PROGRAM SP3_1_Y130
VAR
	CompareOutput130_00: CMP_OC_DW;
	CompareOutput130_01: CMP_OC_DW;
	CompareOutput130_02: CMP_OC_DW;
	CompareOutput130_03: CMP_OC_DW;
	CompareOutput130_04: CMP_OC_DW;
	CompareOutput130_05: CMP_OC_DW;
	CompareOutput130_06: CMP_OC_DW;
	CompareOutput130_07: CMP_OC_DW;
	CompareOutput130_08: CMP_OC_DW;
	CompareOutput130_09: CMP_OC_DW;
	CompareOutput130_10: CMP_OC_DW;
	CompareOutput130_11: CMP_OC_DW;
	CompareOutput130_12: CMP_OC_DW;
	CompareOutput130_13: CMP_OC_DW;
	CompareOutput130_14: CMP_OC_DW;
	CompareOutput130_15: CMP_OC_DW;

END_VAR

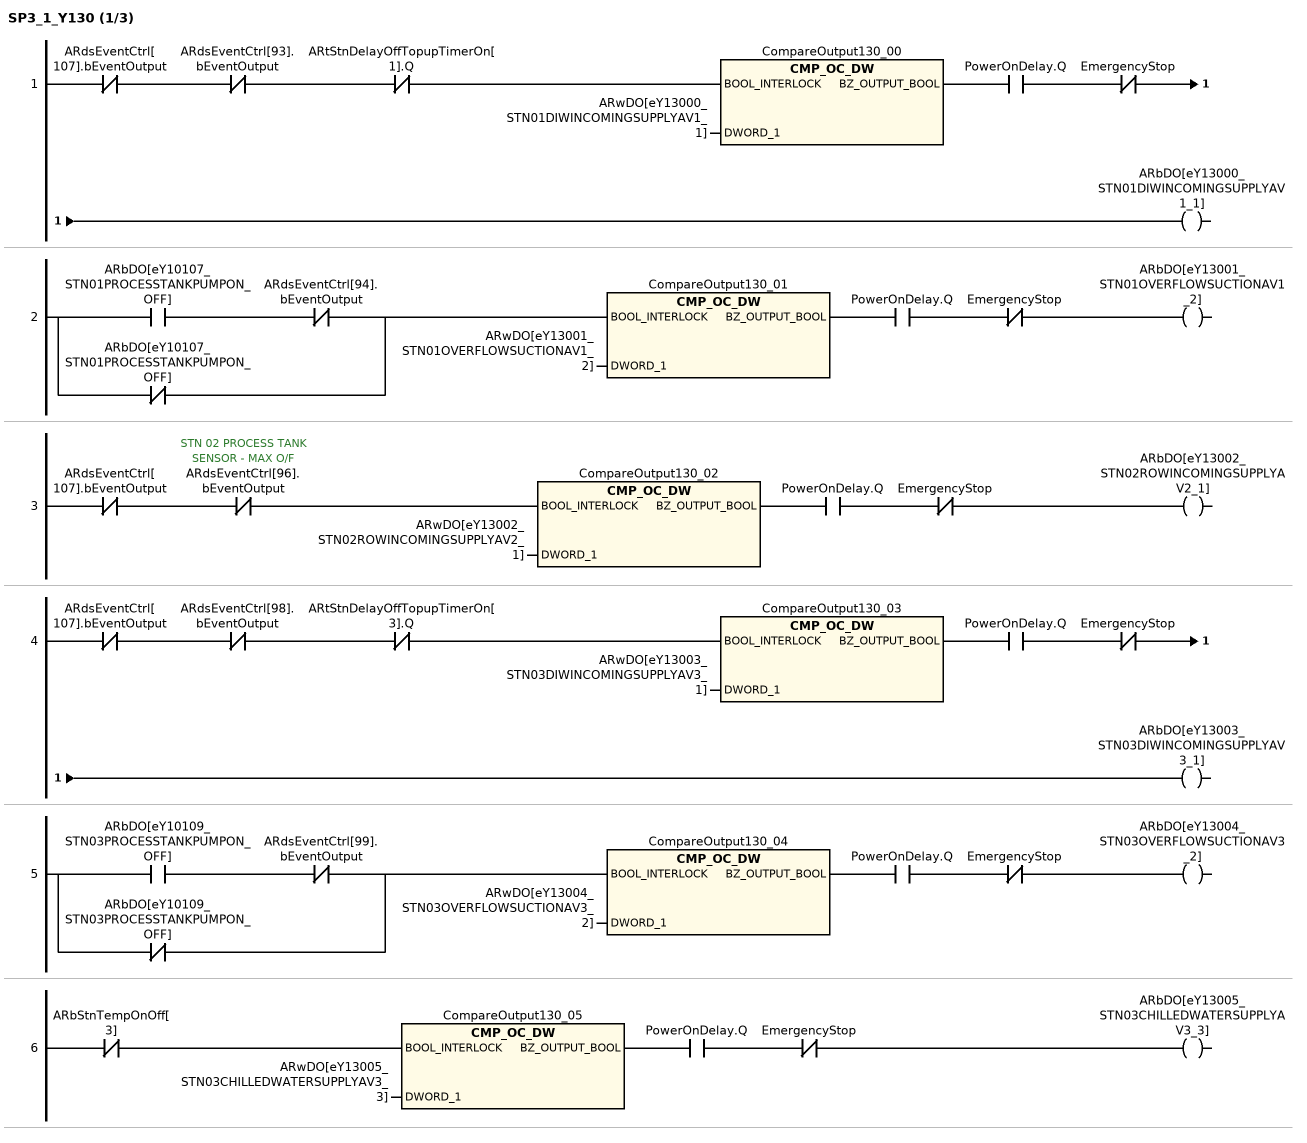
// NETWORK 1
CompareOutput130_00(BOOL_INTERLOCK := NOT ARdsEventCtrl[107].bEventOutput AND NOT ARdsEventCtrl[93].bEventOutput AND NOT ARtStnDelayOffTopupTimerOn[1].Q, DWORD_1 := ARwDO[eY13000_STN01DIWINCOMINGSUPPLYAV1_1]); // CMP_OC_DW
ARbDO[eY13000_STN01DIWINCOMINGSUPPLYAV1_1] := CompareOutput130_00.BZ_OUTPUT_BOOL AND PowerOnDelay.Q AND NOT EmergencyStop;

// NETWORK 2
CompareOutput130_01(BOOL_INTERLOCK := ARbDO[eY10107_STN01PROCESSTANKPUMPON_OFF] AND NOT ARdsEventCtrl[94].bEventOutput OR NOT ARbDO[eY10107_STN01PROCESSTANKPUMPON_OFF], DWORD_1 := ARwDO[eY13001_STN01OVERFLOWSUCTIONAV1_2]); // CMP_OC_DW
ARbDO[eY13001_STN01OVERFLOWSUCTIONAV1_2] := CompareOutput130_01.BZ_OUTPUT_BOOL AND PowerOnDelay.Q AND NOT EmergencyStop;

// NETWORK 3
//   ARdsEventCtrl[96].bEventOutput: STN 02 PROCESS TANK SENSOR - MAX O/F
CompareOutput130_02(BOOL_INTERLOCK := NOT ARdsEventCtrl[107].bEventOutput AND NOT ARdsEventCtrl[96].bEventOutput, DWORD_1 := ARwDO[eY13002_STN02ROWINCOMINGSUPPLYAV2_1]); // CMP_OC_DW
ARbDO[eY13002_STN02ROWINCOMINGSUPPLYAV2_1] := CompareOutput130_02.BZ_OUTPUT_BOOL AND PowerOnDelay.Q AND NOT EmergencyStop;

// NETWORK 4
CompareOutput130_03(BOOL_INTERLOCK := NOT ARdsEventCtrl[107].bEventOutput AND NOT ARdsEventCtrl[98].bEventOutput AND NOT ARtStnDelayOffTopupTimerOn[3].Q, DWORD_1 := ARwDO[eY13003_STN03DIWINCOMINGSUPPLYAV3_1]); // CMP_OC_DW
ARbDO[eY13003_STN03DIWINCOMINGSUPPLYAV3_1] := CompareOutput130_03.BZ_OUTPUT_BOOL AND PowerOnDelay.Q AND NOT EmergencyStop;

// NETWORK 5
CompareOutput130_04(BOOL_INTERLOCK := ARbDO[eY10109_STN03PROCESSTANKPUMPON_OFF] AND NOT ARdsEventCtrl[99].bEventOutput OR NOT ARbDO[eY10109_STN03PROCESSTANKPUMPON_OFF], DWORD_1 := ARwDO[eY13004_STN03OVERFLOWSUCTIONAV3_2]); // CMP_OC_DW
ARbDO[eY13004_STN03OVERFLOWSUCTIONAV3_2] := CompareOutput130_04.BZ_OUTPUT_BOOL AND PowerOnDelay.Q AND NOT EmergencyStop;

// NETWORK 6
CompareOutput130_05(BOOL_INTERLOCK := NOT ARbStnTempOnOff[3], DWORD_1 := ARwDO[eY13005_STN03CHILLEDWATERSUPPLYAV3_3]); // CMP_OC_DW
ARbDO[eY13005_STN03CHILLEDWATERSUPPLYAV3_3] := CompareOutput130_05.BZ_OUTPUT_BOOL AND PowerOnDelay.Q AND NOT EmergencyStop;

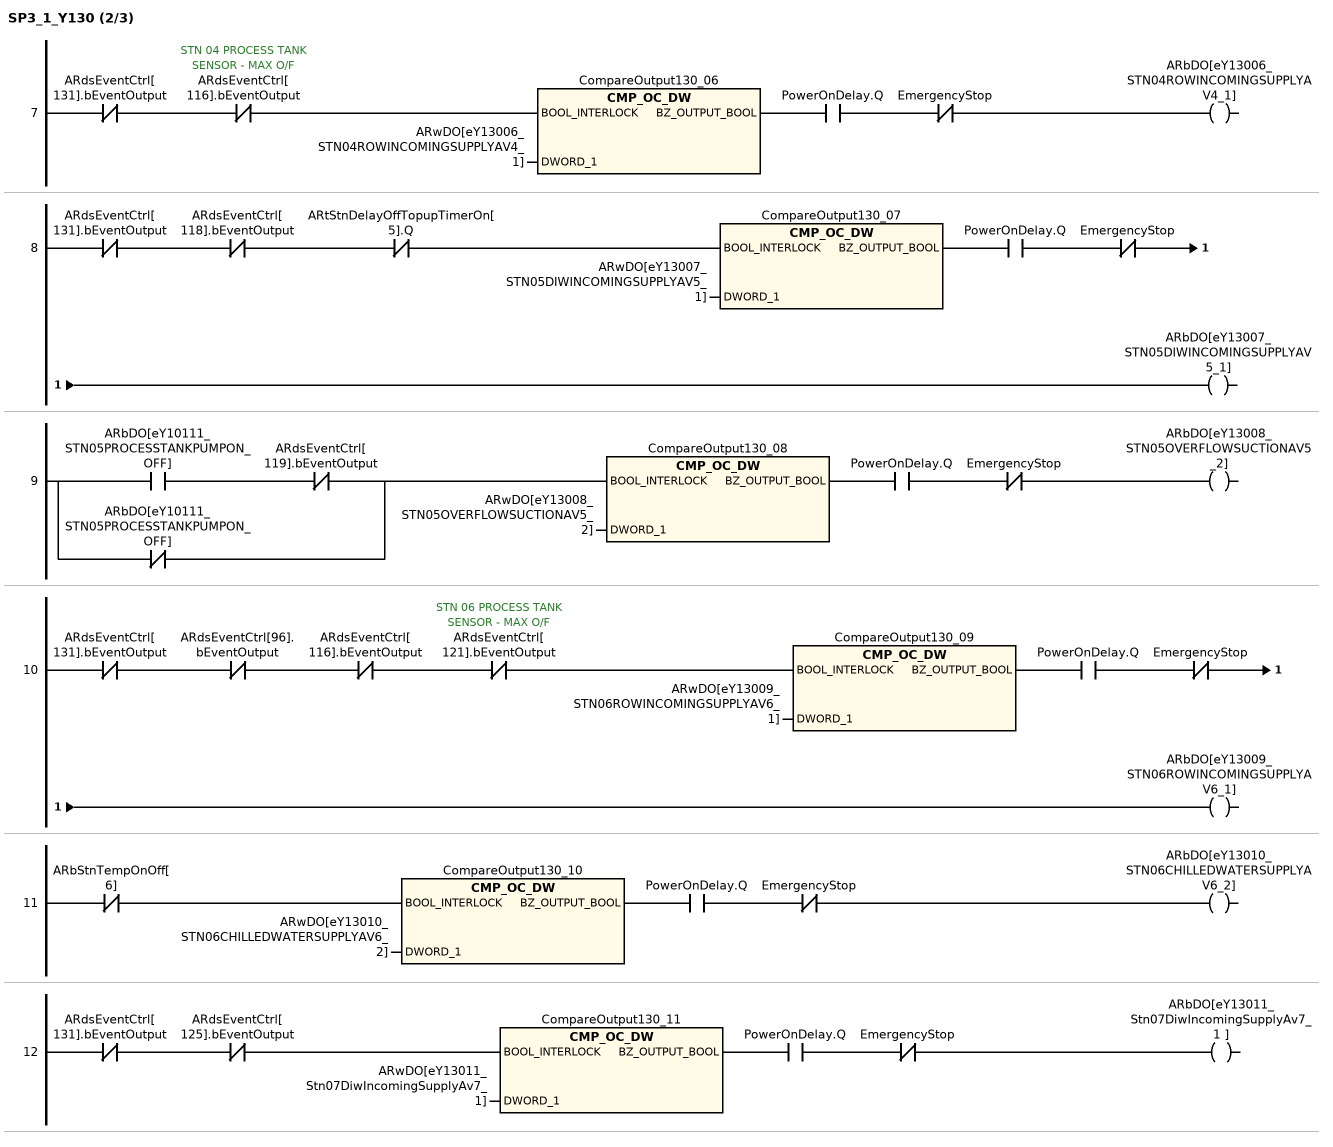
// NETWORK 7
//   ARdsEventCtrl[116].bEventOutput: STN 04 PROCESS TANK SENSOR - MAX O/F
CompareOutput130_06(BOOL_INTERLOCK := NOT ARdsEventCtrl[131].bEventOutput AND NOT ARdsEventCtrl[116].bEventOutput, DWORD_1 := ARwDO[eY13006_STN04ROWINCOMINGSUPPLYAV4_1]); // CMP_OC_DW
ARbDO[eY13006_STN04ROWINCOMINGSUPPLYAV4_1] := CompareOutput130_06.BZ_OUTPUT_BOOL AND PowerOnDelay.Q AND NOT EmergencyStop;

// NETWORK 8
CompareOutput130_07(BOOL_INTERLOCK := NOT ARdsEventCtrl[131].bEventOutput AND NOT ARdsEventCtrl[118].bEventOutput AND NOT ARtStnDelayOffTopupTimerOn[5].Q, DWORD_1 := ARwDO[eY13007_STN05DIWINCOMINGSUPPLYAV5_1]); // CMP_OC_DW
ARbDO[eY13007_STN05DIWINCOMINGSUPPLYAV5_1] := CompareOutput130_07.BZ_OUTPUT_BOOL AND PowerOnDelay.Q AND NOT EmergencyStop;

// NETWORK 9
CompareOutput130_08(BOOL_INTERLOCK := ARbDO[eY10111_STN05PROCESSTANKPUMPON_OFF] AND NOT ARdsEventCtrl[119].bEventOutput OR NOT ARbDO[eY10111_STN05PROCESSTANKPUMPON_OFF], DWORD_1 := ARwDO[eY13008_STN05OVERFLOWSUCTIONAV5_2]); // CMP_OC_DW
ARbDO[eY13008_STN05OVERFLOWSUCTIONAV5_2] := CompareOutput130_08.BZ_OUTPUT_BOOL AND PowerOnDelay.Q AND NOT EmergencyStop;

// NETWORK 10
//   ARdsEventCtrl[121].bEventOutput: STN 06 PROCESS TANK SENSOR - MAX O/F
CompareOutput130_09(BOOL_INTERLOCK := NOT ARdsEventCtrl[131].bEventOutput AND NOT ARdsEventCtrl[96].bEventOutput AND NOT ARdsEventCtrl[116].bEventOutput AND NOT ARdsEventCtrl[121].bEventOutput, DWORD_1 := ARwDO[eY13009_STN06ROWINCOMINGSUPPLYAV6_1]); // CMP_OC_DW
ARbDO[eY13009_STN06ROWINCOMINGSUPPLYAV6_1] := CompareOutput130_09.BZ_OUTPUT_BOOL AND PowerOnDelay.Q AND NOT EmergencyStop;

// NETWORK 11
CompareOutput130_10(BOOL_INTERLOCK := NOT ARbStnTempOnOff[6], DWORD_1 := ARwDO[eY13010_STN06CHILLEDWATERSUPPLYAV6_2]); // CMP_OC_DW
ARbDO[eY13010_STN06CHILLEDWATERSUPPLYAV6_2] := CompareOutput130_10.BZ_OUTPUT_BOOL AND PowerOnDelay.Q AND NOT EmergencyStop;

// NETWORK 12
CompareOutput130_11(BOOL_INTERLOCK := NOT ARdsEventCtrl[131].bEventOutput AND NOT ARdsEventCtrl[125].bEventOutput, DWORD_1 := ARwDO[eY13011_Stn07DiwIncomingSupplyAv7_1]); // CMP_OC_DW
ARbDO[eY13011_Stn07DiwIncomingSupplyAv7_1 ] := CompareOutput130_11.BZ_OUTPUT_BOOL AND PowerOnDelay.Q AND NOT EmergencyStop;

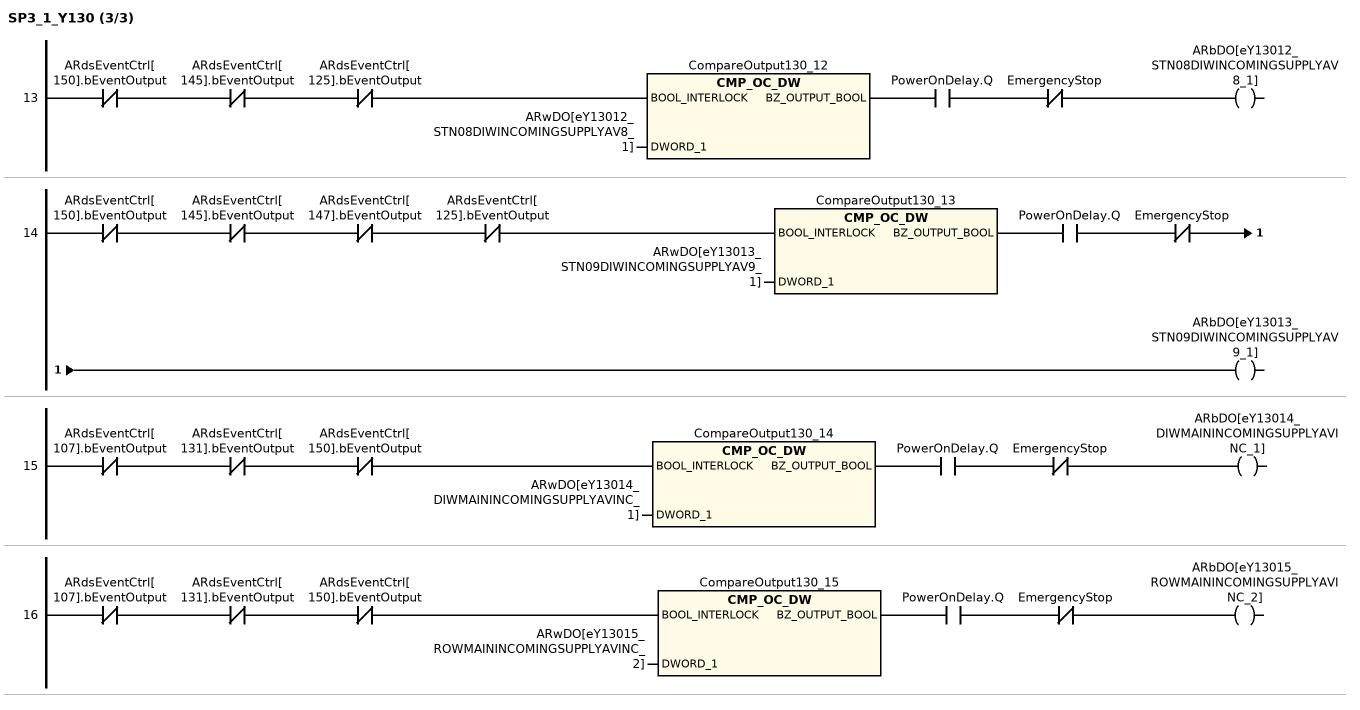
// NETWORK 13
CompareOutput130_12(BOOL_INTERLOCK := NOT ARdsEventCtrl[150].bEventOutput AND NOT ARdsEventCtrl[145].bEventOutput AND NOT ARdsEventCtrl[125].bEventOutput, DWORD_1 := ARwDO[eY13012_STN08DIWINCOMINGSUPPLYAV8_1]); // CMP_OC_DW
ARbDO[eY13012_STN08DIWINCOMINGSUPPLYAV8_1] := CompareOutput130_12.BZ_OUTPUT_BOOL AND PowerOnDelay.Q AND NOT EmergencyStop;

// NETWORK 14
CompareOutput130_13(BOOL_INTERLOCK := NOT ARdsEventCtrl[150].bEventOutput AND NOT ARdsEventCtrl[145].bEventOutput AND NOT ARdsEventCtrl[147].bEventOutput AND NOT ARdsEventCtrl[125].bEventOutput, DWORD_1 := ARwDO[eY13013_STN09DIWINCOMINGSUPPLYAV9_1]); // CMP_OC_DW
ARbDO[eY13013_STN09DIWINCOMINGSUPPLYAV9_1] := CompareOutput130_13.BZ_OUTPUT_BOOL AND PowerOnDelay.Q AND NOT EmergencyStop;

// NETWORK 15
CompareOutput130_14(BOOL_INTERLOCK := NOT ARdsEventCtrl[107].bEventOutput AND NOT ARdsEventCtrl[131].bEventOutput AND NOT ARdsEventCtrl[150].bEventOutput, DWORD_1 := ARwDO[eY13014_DIWMAININCOMINGSUPPLYAVINC_1]); // CMP_OC_DW
ARbDO[eY13014_DIWMAININCOMINGSUPPLYAVINC_1] := CompareOutput130_14.BZ_OUTPUT_BOOL AND PowerOnDelay.Q AND NOT EmergencyStop;

// NETWORK 16
CompareOutput130_15(BOOL_INTERLOCK := NOT ARdsEventCtrl[107].bEventOutput AND NOT ARdsEventCtrl[131].bEventOutput AND NOT ARdsEventCtrl[150].bEventOutput, DWORD_1 := ARwDO[eY13015_ROWMAININCOMINGSUPPLYAVINC_2]); // CMP_OC_DW
ARbDO[eY13015_ROWMAININCOMINGSUPPLYAVINC_2] := CompareOutput130_15.BZ_OUTPUT_BOOL AND PowerOnDelay.Q AND NOT EmergencyStop;

END_PROGRAM

(* stored: Version 1.1.0.1, ProductVersion 3.1.4024.11
   POU SP3_1_Y130: Id {44f2397b-27d6-497d-988d-29d163b30af3}, SpecialFunc None *)
